// SIMATIC S7-200 project (STEP 7-Micro/WIN), CPU 221 REL 01.10

SYMBOL_TABLE USER1
start            I0.0
estop            I0.1
dc               Q0.0
END_SYMBOL_TABLE

ORGANIZATION_BLOCK MAIN:OB1
TITLE=PROGRAM COMMENTS
BEGIN
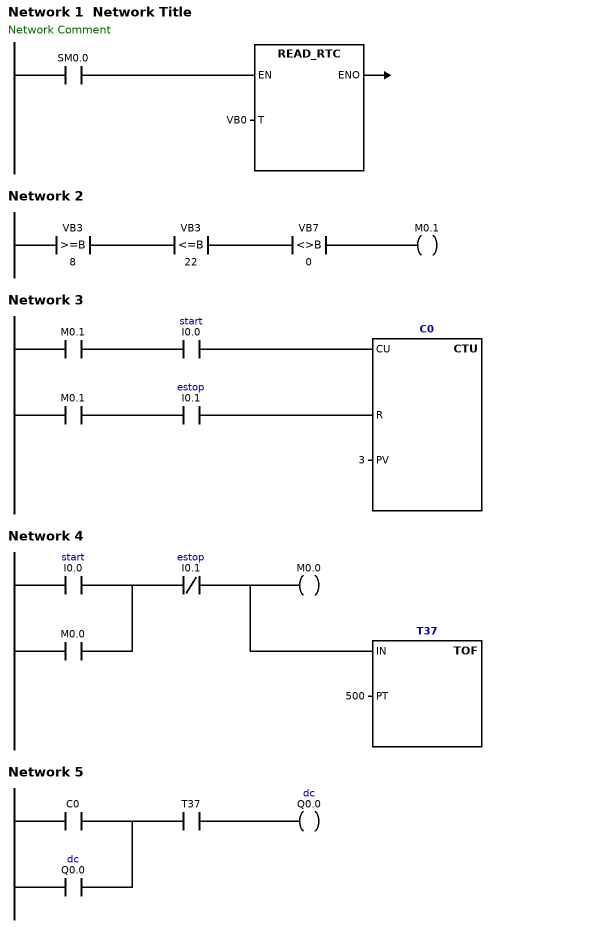
Network 1 // Network Title
// Network Comment
LD     SM0.0
TODR   VB0
Network 2
LDB>=  VB3, 8
AB<=   VB3, 22
AB<>   VB7, 0
=      M0.1
Network 3
LD     M0.1
A      start:I0.0
LD     M0.1
A      estop:I0.1
CTU    C0, 3
Network 4
LD     start:I0.0
O      M0.0
AN     estop:I0.1
=      M0.0
TOF    T37, 500
Network 5
LD     C0
O      dc:Q0.0
A      T37
=      dc:Q0.0
END_ORGANIZATION_BLOCK
